{attribute 'GeneratedUsingTerminal: EK1122-0000-0018'}
{attribute addProperty BoxType "EK1122-0000-0018"}
{attribute addProperty Id "RP10_VI_AES_D_BC_ECAT_xAES_B47A261080RP10_SAFETY_Flexi_Soft_EtherCAT_GatewayFlexi_Soft_EtherCAT_Gateway_DE394EDD5RP10_AB0_EPP1322_0001EPP1322_1FC0878B2RP10_AB1_EPP1008_0001EPP1008_78E8D3DD12RP10_AB2_EPP1008_0001EPP1008_78E8D3DD12RP10_AB3_EPP1008_0001EPP1008_78E8D3DD12RP10_AB4_EPP1008_0001EPP1008_78E8D3DD12"}
{attribute addProperty CRC "1437375578"}
{attribute addProperty Size "135"}
{attribute addProperty Name "RP10_A2 (EK1122)"}
TYPE RP10_A2_EK1122_55AC9C5A EXTENDS EK1122_1FC0878B :
STRUCT
	{attribute addProperty Name "RP10-VI (AES-D-BC-ECAT)"}
	{attribute addProperty PreviousPort "RP10_A2 (EK1122) : D"}
	{attribute addProperty SyncUnit "P10"}
	RP10_VI_AES_D_BC_ECAT_x : AES_B47A2610;
	{attribute addProperty Name "RP10-SAFETY (Flexi Soft EtherCAT Gateway)"}
	{attribute addProperty PreviousPort "RP10_A2 (EK1122) : B"}
	{attribute addProperty SyncUnit "P10"}
	RP10_SAFETY_Flexi_Soft_EtherCAT_Gateway : Flexi_Soft_EtherCAT_Gateway_DE394EDD;
	{attribute addProperty Name "RP10-AB0 (EPP1322-0001)"}
	{attribute addProperty PreviousPort "RP10-SAFETY (Flexi Soft EtherCAT Gateway) : B"}
	{attribute addProperty SyncUnit "default"}
	RP10_AB0_EPP1322_0001 : EPP1322_1FC0878B;
	{attribute addProperty Name "RP10-AB1 (EPP1008-0001)"}
	{attribute addProperty PreviousPort "RP10-AB0 (EPP1322-0001) : C"}
	{attribute addProperty SyncUnit "P10"}
	RP10_AB1_EPP1008_0001 : EPP1008_78E8D3DD;
	{attribute addProperty Name "RP10-AB2 (EPP1008-0001)"}
	{attribute addProperty PreviousPort "RP10-AB1 (EPP1008-0001) : B"}
	{attribute addProperty SyncUnit "P10"}
	RP10_AB2_EPP1008_0001 : EPP1008_78E8D3DD;
	{attribute addProperty Name "RP10-AB3 (EPP1008-0001)"}
	{attribute addProperty PreviousPort "RP10-AB2 (EPP1008-0001) : B"}
	{attribute addProperty SyncUnit "P10"}
	RP10_AB3_EPP1008_0001 : EPP1008_78E8D3DD;
	{attribute addProperty Name "RP10-AB4 (EPP1008-0001)"}
	{attribute addProperty PreviousPort "RP10-AB3 (EPP1008-0001) : B"}
	{attribute addProperty SyncUnit "P10"}
	RP10_AB4_EPP1008_0001 : EPP1008_78E8D3DD;
END_STRUCT
END_TYPE

(* stored: Version 1.2.0.0, ProductVersion 3.1.4024.11
   DUT RP10_A2_EK1122_55AC9C5A: Id {d73998bc-6a24-0d12-0f20-e50659d5add2} *)
